FUNCTION_BLOCK FB_SimulatedHeater EXTENDS FB_ComponentBase IMPLEMENTS I_HeatingElement
VAR
	_Power : BOOL;
END_VAR

{warning 'Add method implementation '}
METHOD CyclicLogic
END_METHOD

PROPERTY Power : BOOL
GET
Power := _Power;
END_GET
END_PROPERTY

METHOD PowerOff : BOOL
_Power := FALSE;
END_METHOD

METHOD PowerOn : BOOL
_Power := TRUE;
END_METHOD

END_FUNCTION_BLOCK

(* stored: Version 1.1.0.1
   POU FB_SimulatedHeater: Id {207790fd-1039-4a93-8685-793b58035a9b}, SpecialFunc None
   Method CyclicLogic: Id {773e2fea-8528-462f-92f6-998c6a861586}
   Property Power: Id {3a4101b8-7c16-4ca6-96b7-cb44bedcc000}
   Get Get: Id {e40ba655-cb2c-4762-9d5e-3363a1e416b3}
   Method PowerOff: Id {0812bacd-6794-4d57-af03-e0437fcc0d00}
   Method PowerOn: Id {a8d9e76d-caf9-41c4-9b20-5070584fb945} *)
